TYPE (* Actuator target states: Work1/Work2/Home *)
  (* Standard: 1131-3 *)
  (* Version 0.1, 6/21/2026, easensoy, WMG, single STRUCT input wrapping the target states *)
  PACKAGE Main;
  TargetStates : STRUCT
    Work1 : INT;
    Work2 : INT;
    Home : INT;
  END_STRUCT;
END_TYPE
